// TIA Portal V17 export
// export: Created 2024-08-09T12:53:18.4506307Z, ExportSetting WithDefaults, DisplayName Totally Integrated Automation Portal, DisplayVersion V17 Update 7, DisplayName TIA Portal Openness, DisplayVersion V17 Update 7, DisplayName TIA Portal Version Control Interface, DisplayVersion V17, DisplayName STEP 7 Professional, DisplayVersion V17 Update 7, DisplayName STEP 7 Safety, DisplayVersion V17 Update 6, DisplayName WinCC Professional, DisplayVersion V17 Update 7
TYPE "Gproduct"
// stored: IsFailsafeCompliant false
   STRUCT
      Etp : SInt;
      Etp_Memo : SInt := -1;
      Etp_Prec : SInt;
      NumZone : SInt;
      Tps_Picke : Date_And_Time;
      Tempo_Inter_Rech : Time;
      Lst_Taches_Fin_Lot : Array[0..9] of "S_TacheNiv";
      Dial_Def : "S_DIALOG_DEF";
   END_STRUCT;
END_TYPE
